PROGRAM FAST
VAR
	nChan : INT;
	MOS_TS: INT;
END_VAR

(****************************************************************************************)
(*	  							Wait for HLI initialization								*)
(****************************************************************************************)
IF NOT CNCSystem.bHLIInit THEN
	RETURN;
END_IF

(* Programm call for MOS_TS M functions *)
// PRG_FastMFunctions();

END_PROGRAM

(* stored: Version 1.1.0.1, ProductVersion 3.1.4023.8
   POU FAST: Id {16c202d0-b697-4d74-8856-0055624c8fd5}, SpecialFunc None *)
